{attribute addProperty BoxType "EJ1914-0000-0017"}
{attribute addProperty Id "FSOEAT %Q*FSOE_27E40C71486"}
{attribute addProperty CRC "3800498592"}
{attribute addProperty SizeInBites "48"}
{attribute addProperty SizeInBytes "6"}
TYPE FSoE_Outputs_E28701A0 :
STRUCT
	{attribute addProperty Name "FSOE"}
	FSOE AT %Q* : FSOE_27E40C71;
END_STRUCT
END_TYPE

(* stored: Version 1.2.0.0, ProductVersion 3.1.4024.9
   DUT FSoE_Outputs_E28701A0: Id {88b38371-f8a6-456b-956a-a24717e02930} *)
